// TIA Portal V18 export
// export: Created 2026-01-09T11:23:35.7334873Z, ExportSetting WithDefaults, DisplayName Totally Integrated Automation Portal, DisplayVersion V18 Update 5, DisplayName TIA Portal Openness, DisplayVersion V18 Update 5, DisplayName TIA Portal Teamcenter Gateway, DisplayVersion V18, DisplayName TIA Portal Version Control Interface, DisplayVersion V18, DisplayName SINAMICS Startdrive Advanced, DisplayVersion V18 SP2 Update 1, DisplayName SINAMICS Startdrive G110M, G120, G120C, G120D, G120P, G115D, DisplayVersion V18 SP2 Update 1, DisplayName SINAMICS Startdrive G130, G150, S120, S150, SINAMICS MV, S210, G220, S200, DisplayVersion V18 SP2 Update 1, DisplayName STEP 7 Professional, DisplayVersion V18 Update 5, DisplayName STEP 7 Safety, DisplayVersion V18, DisplayName WinCC Professional, DisplayVersion V18 Update 5
Screen "274_Motor_J2"  1280x800, Number=274, Template=02ManualUnit1
  ScreenLayer "Layer_0"
    Button "btnMenu5" at 512,725 size 128x75  Mode=Text, TextOff="J-电机2 / J-Motor2", TextOn="J-电机2 / J-Motor2"
      on Click: ActivateScreen(Screen name := , Object number := 0)
    FaceplateInstance "Motor_1" at 70,138 size 273x159  FaceplateTypeName=03 FunctionBlocks@$@202 Conveyer_Line@$@202.2 HMI@$@Motor V 0.0.9
      MotorControl := MotorControl_Dev{2}
      InterfacePropertyText "TextName"  Text="J_提升电机 / J_Lifting Motor"
    FaceplateInstance "Motor_2" at 370,138 size 273x159  FaceplateTypeName=03 FunctionBlocks@$@202 Conveyer_Line@$@202.2 HMI@$@Motor V 0.0.9
      MotorControl := MotorControl_Dev{13}
      InterfacePropertyText "TextName"  Text="J_Magnet上料电机 / J_MagnetLoadingMotor"
    FaceplateInstance "Motor_3" at 670,138 size 273x159  FaceplateTypeName=03 FunctionBlocks@$@202 Conveyer_Line@$@202.2 HMI@$@Motor V 0.0.9
      MotorControl := MotorControl_Dev{14}
      InterfacePropertyText "TextName"  Text="J_Magnet下料电机 / J_MagnetTakeMotor"
    Button "按钮_9" at 128,725 size 128x75  Mode=Text, PictureOff=向右箭头_0, TextOff="J-气缸1 / J-Cylinder1", TextOn="J-气缸1 / J-Cylinder1"
      on Click: ActivateScreen(Screen name := 270_Cylinder_J1, Object number := 0)
    Button "btnMenu4" at 384,725 size 128x75  Mode=Text, TextOff="J-气缸2 / J-Cylinder2", TextOn="J-气缸2 / J-Cylinder2"
      on Click: ActivateScreen(Screen name := 273_Cylinder_J2, Object number := 0)
    Button "btnMenu6" at 640,725 size 128x75  Mode=Text, TextOff="J-气缸3 / J-Cylinder3", TextOn="J-气缸3 / J-Cylinder3"
      on Click: ActivateScreen(Screen name := 276_Cylinder_J3, Object number := 0)
    Button "btnMenu7" at 896,725 size 128x75  Mode=Text
    Button "btnMenu6_1" at 768,725 size 128x75  Mode=Text, TextOff="J-电机3 / J-Motor3", TextOn="J-电机3 / J-Motor3"
      on Click: ActivateScreen(Screen name := 277_Motor_J3, Object number := 0)
    Button "btnMenu7_1" at 1024,725 size 128x75  Mode=Text
    Button "btnMenu4_1" at 256,725 size 128x75  Mode=Text, TextOff="J-电机1 / J-Motor1", TextOn="J-电机1 / J-Motor1"
      on Click: ActivateScreen(Screen name := 271_Motor_J1, Object number := 0)
